FUNCTION ARR08B_TO_ST08B
  (* Standard: 61499-1; Description: Copyright (c) 2024 HR Agrartechnik GmbH This program and the accompanying materials are made available under the terms of the Eclipse Public License 2.0 which is available at https://www.eclipse.org/legal/epl-2.0/ SPDX-License-Identifier: EPL-2.0 *)
  (* Version 1.0, 2024-02-22, Franz Höpfinger, HR Agrartechnik GmbH *)
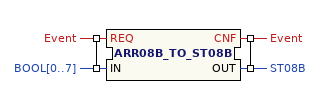
  EVENT_INPUT
    REQ WITH IN; (* Normal Execution Request *)
  END_EVENT
  EVENT_OUTPUT
    CNF WITH OUT; (* Execution Confirmation *)
  END_EVENT
  VAR_INPUT
    IN : ARRAY [0..7] OF BOOL; (* ARR08B Input *)
  END_VAR
  VAR_OUTPUT
    OUT : ST08B; (* ST08B Output *)
  END_VAR
  BODY IN ST:
FUNCTION ARR08B_TO_ST08B

VAR_INPUT
	IN : ARRAY[0..7] OF BOOL;    // ARR08B Input
END_VAR

VAR_OUTPUT
	OUT : ST08B;    // ST08B Output
END_VAR

(* this Function extracts the 8 BOOLS from a byte *)
OUT.B_00 := IN[0];
OUT.B_01 := IN[1];
OUT.B_02 := IN[2];
OUT.B_03 := IN[3];
OUT.B_04 := IN[4];
OUT.B_05 := IN[5];
OUT.B_06 := IN[6];
OUT.B_07 := IN[7];

END_FUNCTION
  END_BODY
END_FUNCTION
